(*			
	RafalOS
	Rafał Osajda		20.11.2025		TC 4024.66
	Moduł przygotowania danych dla Okna głównego w trybie mycia
*)
FUNCTION_BLOCK FB_MCHMIPrepareDataForScreen_00_04 EXTENDS FB_MCHMIPrepareDataForScreen IMPLEMENTS ITF_MCHMIPrepareDataForScreen
VAR
	itfMachineControlHMI	: ITF_MCHMIMachineControl_HMI_PrepScr_00_04;
	refstData				: REFERENCE TO ST_MCHMIPrepareScreen_00_04;
END_VAR

(*			
	RafalOS
	Rafał Osajda		19.11.2025		TC 4024.66
	Czyści danych przy zmienia ramki po poprzedniej ramce
*)
METHOD PUBLIC ClearAfterScreen : BOOL
VAR_INPUT
END_VAR
SUPER^.ClearAfterScreen ();
END_METHOD

METHOD PUBLIC LinkDataHMI_00_04 : BOOL
VAR_INPUT
	refstData				: REFERENCE TO ST_MCHMIPrepareScreen_00_04;
END_VAR
THIS^.refstData REF= refstData;
END_METHOD

METHOD PUBLIC LinkMachineControlHMI : BOOL
VAR_INPUT
	fbMachineControlHMI	: ITF_MCHMIMachineControl_HMI_PrepScr_00_04;
END_VAR
this^.itfMachineControlHMI := fbMachineControlHMI;
END_METHOD

(*			
	RafalOS
	Rafał Osajda		14.11.2025		TC 4024.66
	Metoda przygotowywania danych dla HMI 
	W niej odbywa się odpytywanie właściego elementu przez łącznik
*)
METHOD PUBLIC PrepareDataForHMI : BOOL
VAR_INPUT
END_VAR
SUPER^.PrepareDataForHMI ();
END_METHOD

(*			
	RafalOS
	Rafał Osajda		19.11.2025		TC 4024.66
	Przygotowanie ramki pood tamke do wyświetlenia - tylko przygotowanie a nie przygotowanie danych do wyświetlenia
*)
METHOD PUBLIC PrepareForScreen : BOOL
VAR_INPUT
END_VAR
SUPER^.PrepareForScreen ();
END_METHOD

END_FUNCTION_BLOCK

(* stored: Version 1.1.0.1
   POU FB_MCHMIPrepareDataForScreen_00_04: Id {6aec6ede-830d-0b83-322c-98ba6a94cacb}, SpecialFunc None
   Folder ITF_PDFS: Id {10397e43-8ded-0db6-3620-9499aec0667f}
   Method ClearAfterScreen: Id {57e6c74e-82cc-0576-14a6-28f6c01fcd38}
   Method LinkDataHMI_00_04: Id {48d968b0-bbda-024b-2f1e-a241eb06fa92}
   Method LinkMachineControlHMI: Id {28da5b0d-943a-0b57-205a-30f22ee9175b}
   Method PrepareDataForHMI: Id {9fd8f0d6-6988-002a-0536-48fe775011e8}
   Method PrepareForScreen: Id {fd55314e-995d-0e12-0095-ce1375d32db3} *)
